TYPE ICode : 
STRUCT
	bComOpen:BOOL;  //扫码Tcp 开
    bComClose:BOOL;  //扫码Tcp 关

	bLON :BOOL; //  扫码开
	bLOFF :BOOL; //扫码关
	bDone  :BOOL; //扫码完成
    bError :BOOL;//扫码故障	
    strCode:STRING;//条码结果
    bCodeConError:BOOL;
END_STRUCT
END_TYPE

(* stored: Version 1.1.0.1, ProductVersion 3.1.4024.9
   DUT ICode: Id {6f2d76e9-8c21-4e81-9e2b-5d28f0256491} *)
